// SIMATIC S7-200 SMART project (STEP 7-Micro/WIN SMART), CPU SR40

SYMBOL_TABLE 表格 1
阀1远程开            V0.0
阀2远程开            V0.1
阀3远程开            V0.2
阀4远程开            V0.3
阀5远程开            V0.4
阀6远程开            V0.5
阀7远程开            V0.6
阀8远程开            V0.7
阀9远程开            V1.0
阀10远程开           V1.1
泵1远程开            V1.2
泵2远程开            V1.3
泵3远程开            V1.4
泵4远程开            V1.5
远程一键开阀           V2.2
远程一键关阀           V2.3
END_SYMBOL_TABLE

SYMBOL_TABLE 系统符号
Always_On        SM0.0    // 始终接通
END_SYMBOL_TABLE

ORGANIZATION_BLOCK MAIN:OB1
TITLE=程序注释
BEGIN
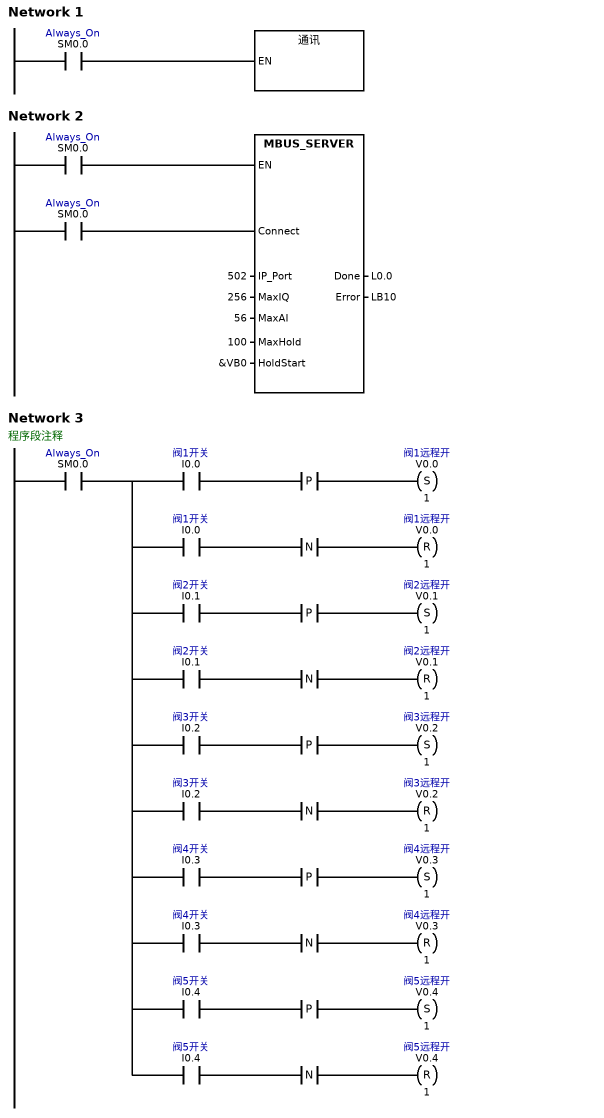
Network 1
LD     Always_On:SM0.0
CALL   通讯:SBR0
Network 2
LD     Always_On:SM0.0
=      L60.0
LD     Always_On:SM0.0
=      L63.7
LD     L60.0
CALL   MBUS_SERVER:SBR6, L63.7, 502, 256, 56, 100, &VB0, L0.0, LB10
Network 3
// 程序段注释
LD     Always_On:SM0.0
LPS
A      阀1开关:I0.0
EU
S      阀1远程开:V0.0, 1
LRD
A      阀1开关:I0.0
ED
R      阀1远程开:V0.0, 1
LRD
A      阀2开关:I0.1
EU
S      阀2远程开:V0.1, 1
LRD
A      阀2开关:I0.1
ED
R      阀2远程开:V0.1, 1
LRD
A      阀3开关:I0.2
EU
S      阀3远程开:V0.2, 1
LRD
A      阀3开关:I0.2
ED
R      阀3远程开:V0.2, 1
LRD
A      阀4开关:I0.3
EU
S      阀4远程开:V0.3, 1
LRD
A      阀4开关:I0.3
ED
R      阀4远程开:V0.3, 1
LRD
A      阀5开关:I0.4
EU
S      阀5远程开:V0.4, 1
LPP
A      阀5开关:I0.4
ED
R      阀5远程开:V0.4, 1
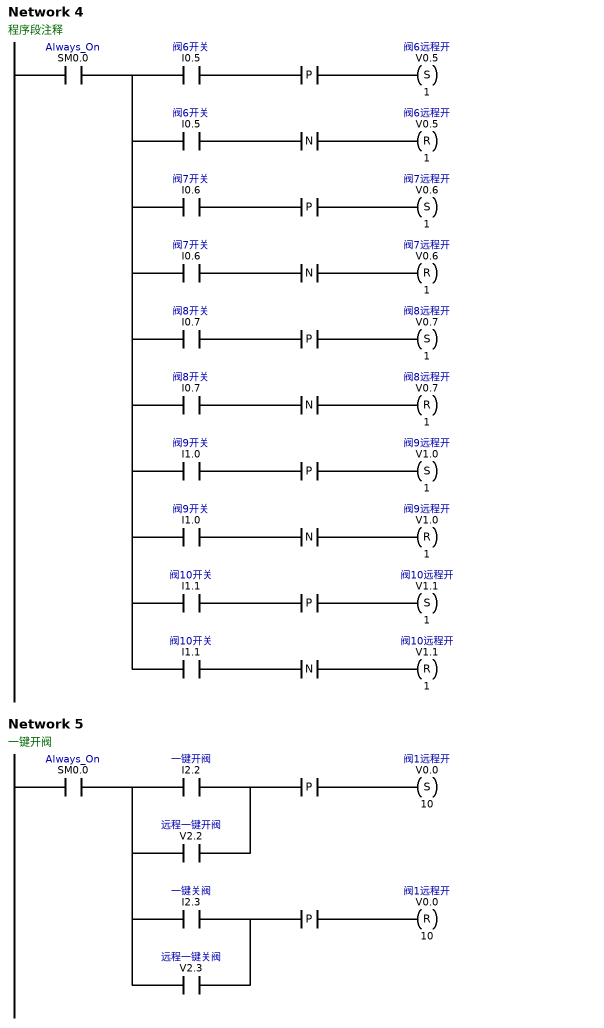
Network 4
// 程序段注释
LD     Always_On:SM0.0
LPS
A      阀6开关:I0.5
EU
S      阀6远程开:V0.5, 1
LRD
A      阀6开关:I0.5
ED
R      阀6远程开:V0.5, 1
LRD
A      阀7开关:I0.6
EU
S      阀7远程开:V0.6, 1
LRD
A      阀7开关:I0.6
ED
R      阀7远程开:V0.6, 1
LRD
A      阀8开关:I0.7
EU
S      阀8远程开:V0.7, 1
LRD
A      阀8开关:I0.7
ED
R      阀8远程开:V0.7, 1
LRD
A      阀9开关:I1.0
EU
S      阀9远程开:V1.0, 1
LRD
A      阀9开关:I1.0
ED
R      阀9远程开:V1.0, 1
LRD
A      阀10开关:I1.1
EU
S      阀10远程开:V1.1, 1
LPP
A      阀10开关:I1.1
ED
R      阀10远程开:V1.1, 1
Network 5
// 一键开阀
LD     Always_On:SM0.0
LPS
LD     一键开阀:I2.2
O      远程一键开阀:V2.2
ALD
EU
S      阀1远程开:V0.0, 10
LPP
LD     一键关阀:I2.3
O      远程一键关阀:V2.3
ALD
EU
R      阀1远程开:V0.0, 10
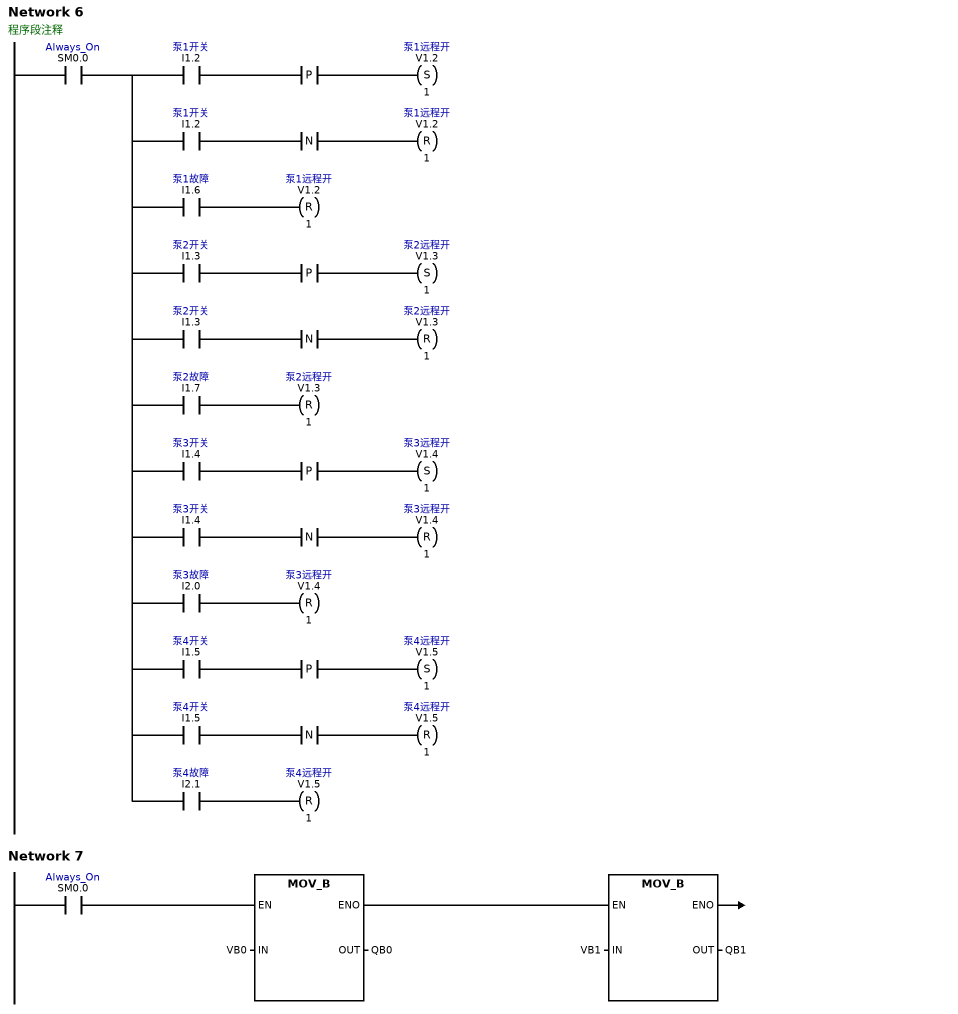
Network 6
// 程序段注释
LD     Always_On:SM0.0
LPS
A      泵1开关:I1.2
EU
S      泵1远程开:V1.2, 1
LRD
A      泵1开关:I1.2
ED
R      泵1远程开:V1.2, 1
LRD
A      泵1故障:I1.6
R      泵1远程开:V1.2, 1
LRD
A      泵2开关:I1.3
EU
S      泵2远程开:V1.3, 1
LRD
A      泵2开关:I1.3
ED
R      泵2远程开:V1.3, 1
LRD
A      泵2故障:I1.7
R      泵2远程开:V1.3, 1
LRD
A      泵3开关:I1.4
EU
S      泵3远程开:V1.4, 1
LRD
A      泵3开关:I1.4
ED
R      泵3远程开:V1.4, 1
LRD
A      泵3故障:I2.0
R      泵3远程开:V1.4, 1
LRD
A      泵4开关:I1.5
EU
S      泵4远程开:V1.5, 1
LRD
A      泵4开关:I1.5
ED
R      泵4远程开:V1.5, 1
LPP
A      泵4故障:I2.1
R      泵4远程开:V1.5, 1
Network 7
LD     Always_On:SM0.0
MOVB   VB0, QB0
AENO
MOVB   VB1, QB1
END_ORGANIZATION_BLOCK

SUBROUTINE_BLOCK 通讯:SBR0
TITLE=子程序注释
BEGIN
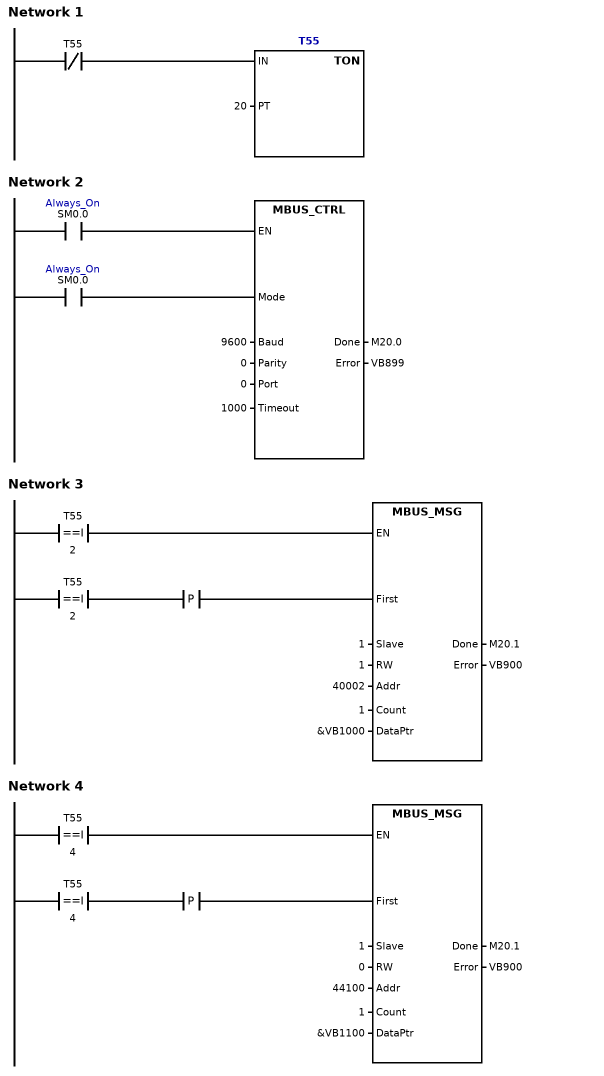
Network 1
LDN    T55
TON    T55, 20
Network 2
LD     Always_On:SM0.0
=      L60.0
LD     Always_On:SM0.0
=      L63.7
LD     L60.0
CALL   MBUS_CTRL:SBR1, L63.7, 9600, 0, 0, 1000, M20.0, VB899
Network 3
LDW=   T55, 2
=      L60.0
LDW=   T55, 2
EU
=      L63.7
LD     L60.0
CALL   MBUS_MSG:SBR2, L63.7, 1, 1, 40002, 1, &VB1000, M20.1, VB900
Network 4
LDW=   T55, 4
=      L60.0
LDW=   T55, 4
EU
=      L63.7
LD     L60.0
CALL   MBUS_MSG:SBR2, L63.7, 1, 0, 44100, 1, &VB1100, M20.1, VB900
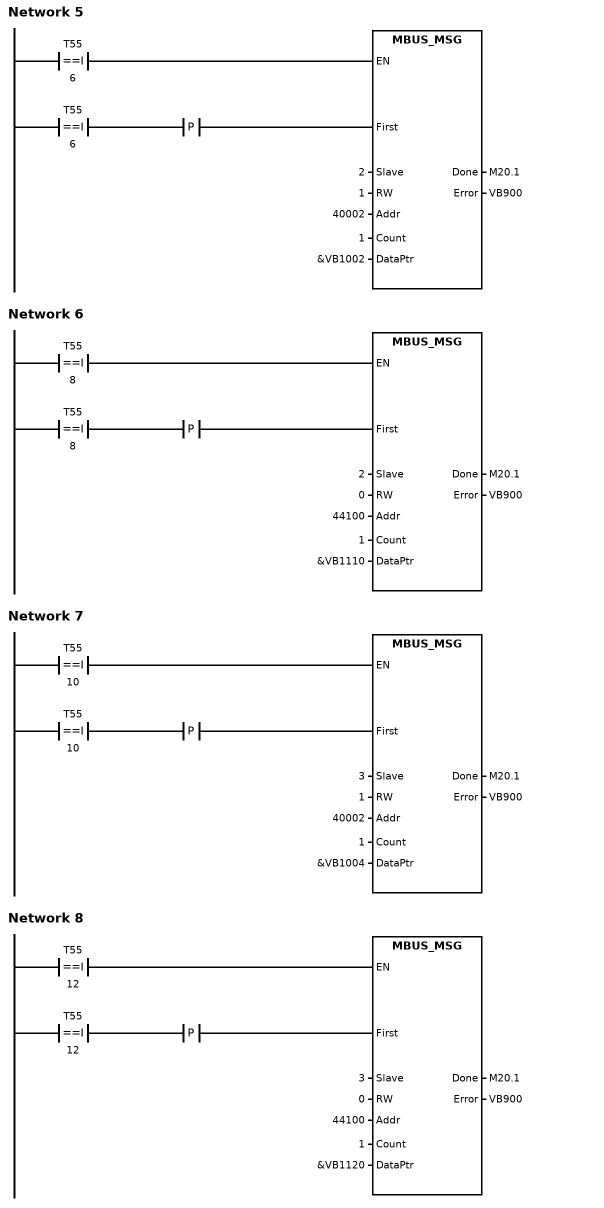
Network 5
LDW=   T55, 6
=      L60.0
LDW=   T55, 6
EU
=      L63.7
LD     L60.0
CALL   MBUS_MSG:SBR2, L63.7, 2, 1, 40002, 1, &VB1002, M20.1, VB900
Network 6
LDW=   T55, 8
=      L60.0
LDW=   T55, 8
EU
=      L63.7
LD     L60.0
CALL   MBUS_MSG:SBR2, L63.7, 2, 0, 44100, 1, &VB1110, M20.1, VB900
Network 7
LDW=   T55, 10
=      L60.0
LDW=   T55, 10
EU
=      L63.7
LD     L60.0
CALL   MBUS_MSG:SBR2, L63.7, 3, 1, 40002, 1, &VB1004, M20.1, VB900
Network 8
LDW=   T55, 12
=      L60.0
LDW=   T55, 12
EU
=      L63.7
LD     L60.0
CALL   MBUS_MSG:SBR2, L63.7, 3, 0, 44100, 1, &VB1120, M20.1, VB900
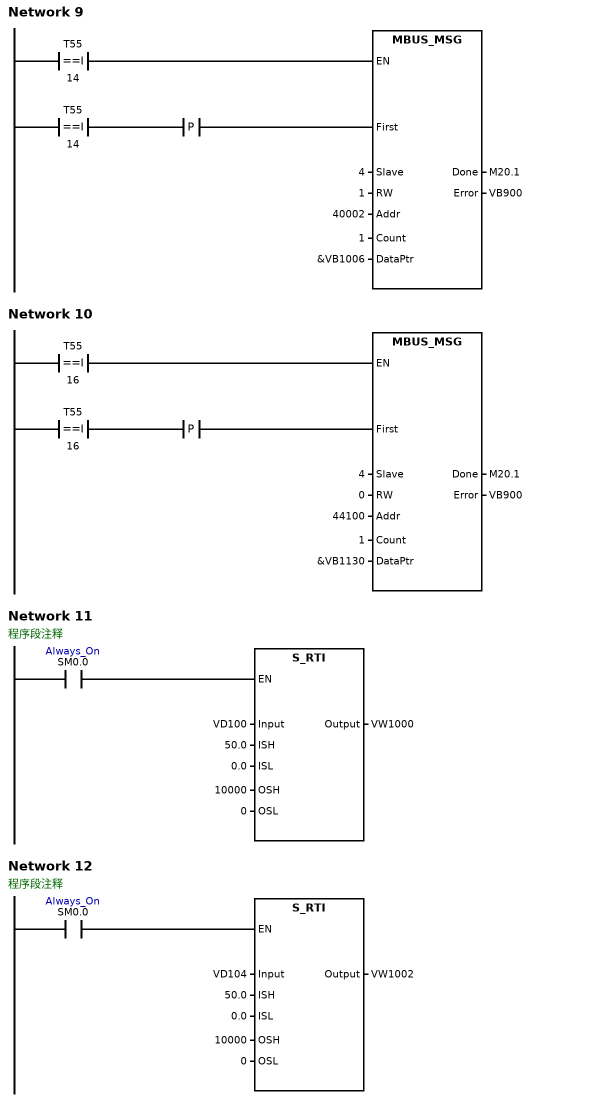
Network 9
LDW=   T55, 14
=      L60.0
LDW=   T55, 14
EU
=      L63.7
LD     L60.0
CALL   MBUS_MSG:SBR2, L63.7, 4, 1, 40002, 1, &VB1006, M20.1, VB900
Network 10
LDW=   T55, 16
=      L60.0
LDW=   T55, 16
EU
=      L63.7
LD     L60.0
CALL   MBUS_MSG:SBR2, L63.7, 4, 0, 44100, 1, &VB1130, M20.1, VB900
Network 11
// 程序段注释
LD     Always_On:SM0.0
CALL   S_RTI:SBR4, VD100, 50.0, 0.0, 10000, 0, VW1000
Network 12
// 程序段注释
LD     Always_On:SM0.0
CALL   S_RTI:SBR4, VD104, 50.0, 0.0, 10000, 0, VW1002
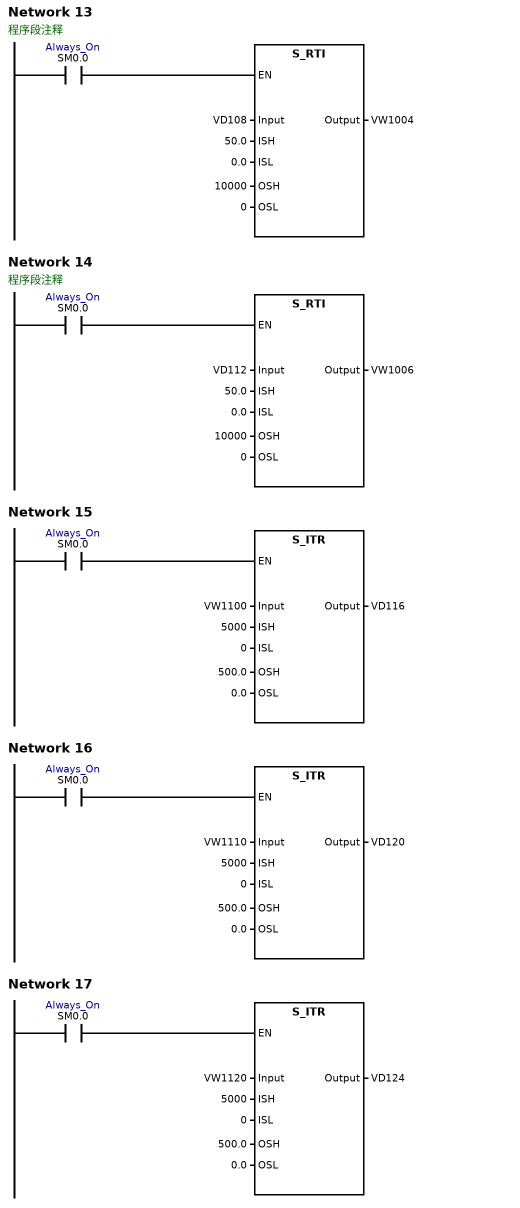
Network 13
// 程序段注释
LD     Always_On:SM0.0
CALL   S_RTI:SBR4, VD108, 50.0, 0.0, 10000, 0, VW1004
Network 14
// 程序段注释
LD     Always_On:SM0.0
CALL   S_RTI:SBR4, VD112, 50.0, 0.0, 10000, 0, VW1006
Network 15
LD     Always_On:SM0.0
CALL   S_ITR:SBR5, VW1100, 5000, 0, 500.0, 0.0, VD116
Network 16
LD     Always_On:SM0.0
CALL   S_ITR:SBR5, VW1110, 5000, 0, 500.0, 0.0, VD120
Network 17
LD     Always_On:SM0.0
CALL   S_ITR:SBR5, VW1120, 5000, 0, 500.0, 0.0, VD124
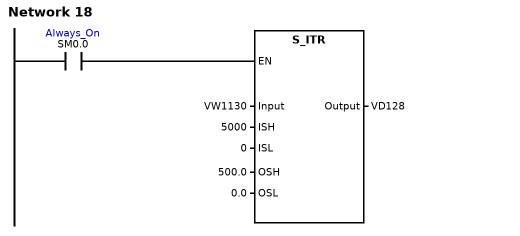
Network 18
LD     Always_On:SM0.0
CALL   S_ITR:SBR5, VW1130, 5000, 0, 500.0, 0.0, VD128
END_SUBROUTINE_BLOCK

// SBR1: protected block, not included

// SBR2: protected block, not included

// SBR3: protected block, not included

// SBR4: protected block, not included

// SBR5: protected block, not included

// SBR6: protected block, not included
